{attribute 'qualified_only'}
VAR_GLOBAL
		stFloorOne	: ST_FloorOne;
END_VAR

(* stored: Version 1.1.0.1, ProductVersion 3.1.4024.12
   GVL House: Id {855b808c-83ef-4d7d-90e8-63f663180320} *)
